// TIA Portal V15.1 export
// export: Created 2020-06-12T07:35:35.6787109Z, ExportSetting None, DisplayName Totally Integrated Automation Portal, DisplayVersion V15.1, DisplayName TIA Portal Openness, DisplayVersion V15.1, DisplayName STEP 7 Professional, DisplayVersion V15.1, DisplayName STEP 7 Safety, DisplayVersion V15.1, DisplayName WinCC Advanced, DisplayVersion V15.1
FUNCTION_BLOCK "RTG1_GLOB_FIO_STATUS"   // FB2, SCL
{ S7_Optimized_Access := 'TRUE' }
// stored: MemoryReserve 100, SetENOAutomatically False
   VAR_OUTPUT
      QSTATUS : Bool;
      RIOforFA_VALUE_STATUS : Bool;
   END_VAR
BEGIN
   #"QSTATUS" := false;
   #"RIOforFA_VALUE_STATUS" := true;
   (*        -K82 | F-DI 8x24VDC HF *)
   #"QSTATUS" := #"QSTATUS" OR ((NOT "F04405_-K82|F-DI8x24VDCHF"."DISABLED") AND ("F04405_-K82|F-DI8x24VDCHF"."QBAD"));
   (*        -K86 | F-DI 8x24VDC HF *)
   #"QSTATUS" := #"QSTATUS" OR ((NOT "F04411_-K86|F-DI8x24VDCHF"."DISABLED") AND ("F04411_-K86|F-DI8x24VDCHF"."QBAD"));
   (* -K102 | F-DQ 4x24VDC/2A PM HF *)
   #"QSTATUS" := #"QSTATUS" OR ((NOT "F04418_-K102|F-DQ4x24VDC/2APMHF"."DISABLED") AND ("F04418_-K102|F-DQ4x24VDC/2APMHF"."QBAD"));
   (*        -K62 | F-DI 8x24VDC HF *)
   #"QSTATUS" := #"QSTATUS" OR ((NOT "F04428_-K62|F-DI8x24VDCHF"."DISABLED") AND ("F04428_-K62|F-DI8x24VDCHF"."QBAD"));
   (*        -K66 | F-DI 8x24VDC HF *)
   #"QSTATUS" := #"QSTATUS" OR ((NOT "F04434_-K66|F-DI8x24VDCHF"."DISABLED") AND ("F04434_-K66|F-DI8x24VDCHF"."QBAD"));
   (*        -K72 | F-DI 8x24VDC HF *)
   #"QSTATUS" := #"QSTATUS" OR ((NOT "F04440_-K72|F-DI8x24VDCHF"."DISABLED") AND ("F04440_-K72|F-DI8x24VDCHF"."QBAD"));
   (*        -K76 | F-DI 8x24VDC HF *)
   #"QSTATUS" := #"QSTATUS" OR ((NOT "F04446_-K76|F-DI8x24VDCHF"."DISABLED") AND ("F04446_-K76|F-DI8x24VDCHF"."QBAD"));
   (*  -K82 | F-DQ 4x24VDC/2A PM HF *)
   #"QSTATUS" := #"QSTATUS" OR ((NOT "F04452_-K82|F-DQ4x24VDC/2APMHF"."DISABLED") AND ("F04452_-K82|F-DQ4x24VDC/2APMHF"."QBAD"));
   (*  -K86 | F-DQ 4x24VDC/2A PM HF *)
   #"QSTATUS" := #"QSTATUS" OR ((NOT "F04457_-K86|F-DQ4x24VDC/2APMHF"."DISABLED") AND ("F04457_-K86|F-DQ4x24VDC/2APMHF"."QBAD"));
   (*  -K92 | F-DQ 4x24VDC/2A PM HF *)
   #"QSTATUS" := #"QSTATUS" OR ((NOT "F04462_-K92|F-DQ4x24VDC/2APMHF"."DISABLED") AND ("F04462_-K92|F-DQ4x24VDC/2APMHF"."QBAD"));
   (*  -K96 | F-DQ 4x24VDC/2A PM HF *)
   #"QSTATUS" := #"QSTATUS" OR ((NOT "F04467_-K96|F-DQ4x24VDC/2APMHF"."DISABLED") AND ("F04467_-K96|F-DQ4x24VDC/2APMHF"."QBAD"));
   (*      -K82 (F-DI 8x24VDC HF_1) *)
   #"QSTATUS" := #"QSTATUS" OR ((NOT "F04476_-K82(F-DI8x24VDCHF_1)"."DISABLED") AND ("F04476_-K82(F-DI8x24VDCHF_1)"."QBAD"));
   #"QSTATUS" := #"QSTATUS" OR NOT #"RIOforFA_VALUE_STATUS";
END_FUNCTION_BLOCK
